// TwinCAT 3 PLC project Operation_Control
// ProgramVersion: 3.1.4023.0
// libraries:
//   Tc2_Standard, * (Beckhoff Automation GmbH)
//   Tc2_System, * (Beckhoff Automation GmbH)
//   Tc3_Module, * (Beckhoff Automation GmbH)
// project tree:
//   DUTs/ OperationControlCommands.TcDUT
//   GVLs/ GVL.TcGVL
//   / PlcTask.TcTTO
//   POUs/ MAIN.TcPOU
// real-time tasks:
//   TASK PlcTask: cycle T#1ms, priority 20, ADS port 350
// I/O:
//   DEVICE Gerät 1 (EtherCAT), AmsNetId 10.183.66.136.2.1
//     Box 1 (CX2040 EtherCAT slave) [CX2040 EtherCAT slave]
// variable links:
//   Operation Control/Operation Control Instance <-> Device 1 (EtherCAT)/Box 1 (CX2040 EtherCAT slave)
//     PlcTask Inputs/GVL.stFromMCToOC <-> IO Inputs/FromMCToOC
//     PlcTask Outputs/GVL.stFromOCToMC <-> IO Outputs/FromOCToMC

CONFIGURATION Operation_Control
    RESOURCE PLC ON TwinCAT3
        TASK PlcTask(INTERVAL := T#1ms, PRIORITY := 20);
        PROGRAM MAIN WITH PlcTask : MAIN;
    END_RESOURCE
END_CONFIGURATION

// ---- DUTs/OperationControlCommands.TcDUT
TYPE OperationControlCommands :
STRUCT
	//Inputs
	bStartOperational 				: BOOL	;
	bStopOperational 				: BOOL	;
	bEndShutdown					: BOOL	;
	bGoToError 						: BOOL	;
	bAckError 						: BOOL	;
	bMinimumAirGapForGC				: BOOL	;
	nOperationMode 					: BYTE	;
	nSafetyCounterOC				: UDINT	;
	
	//Outputs
	bShutdownFinished				: BOOL	;
END_STRUCT
END_TYPE

// ---- GVLs/GVL.TcGVL
{attribute 'qualified_only'}
VAR_GLOBAL
	stFromMCToOC AT %I* : FromMainControlToOperationControl;
	stFromOCToMC AT %Q* : FromOperationControlToMainControl;
END_VAR

// ---- POUs/MAIN.TcPOU
PROGRAM MAIN
VAR
	aIMU0 : ARRAY [0..2] OF REAL;
	aIMU1 : ARRAY [0..2] OF REAL;
	fDistance : REAL;
	
	stCommands : OperationControlCommands;
	bSMDisable : BOOL;
	bLSDisable : BOOL;
	bGSDisable : BOOL;
END_VAR

aIMU0[0] := GVL.stFromMCToOC.MO_origM_GuidanceIMUX0;
aIMU0[1] := GVL.stFromMCToOC.MO_origM_GuidanceIMUY0;
aIMU0[2] := GVL.stFromMCToOC.MO_origM_GuidanceIMUZ0;

aIMU1[0] := GVL.stFromMCToOC.MO_origM_GuidanceIMUX1;
aIMU1[1] := GVL.stFromMCToOC.MO_origM_GuidanceIMUY1;
aIMU1[2] := GVL.stFromMCToOC.MO_origM_GuidanceIMUZ1;

fDistance := GVL.stFromMCToOC.MO_origM_DistanceServiceModule;

GVL.stFromOCToMC.OM_origO_StartOperational := stCommands.bStartOperational;
GVL.stFromOCToMC.OM_origO_StopOperational := stCommands.bStopOperational;
GVL.stFromOCToMC.OM_origO_EndShutdown := stCommands.bEndShutdown;
GVL.stFromOCToMC.OM_origO_GoToError := stCommands.bGoToError;
GVL.stFromOCToMC.OM_origO_AckError := stCommands.bAckError;
GVL.stFromOCToMC.OM_origG_ServiceModuleDisable := bSMDisable;
GVL.stFromOCToMC.OM_origG_LevitationDisable := bLSDisable;
GVL.stFromOCToMC.OM_origG_GuidanceDisable := bGSDisable;

END_PROGRAM
